# EPICS alarm handler configuration: alh_files/mgnt_bsyh.alhConfig
GROUP NULL MGNT:BSYH:1
   $COMMAND edm -x -eolc -noedit mgnt_bsy0_main.edl

$ALIAS BSYH
$GUIDANCE
bsyh Magnet
   Group Name: MGNT:BSYH:1
   Summary PV:  MGNT:BSYH:1:STATSUMY
$END

   INCLUDE MGNT:BSYH:1 ./mgnt_bsyh_lgps.alhConfig
   INCLUDE MGNT:BSYH:1 ./mgnt_bsyh_quad.alhConfig
   INCLUDE MGNT:BSYH:1 ./mgnt_bsyh_xcor.alhConfig
   INCLUDE MGNT:BSYH:1 ./mgnt_bsyh_ycor.alhConfig
